(* CODESYS project SeminarskiV2.project
   Title: SeminarskiV1
   Version: 0.0.0.0

Project tree, tasks and I/O mapping:
  MyController : TM241CE24T/U, Schneider Electric, order no. TM241CE24T/U, version 4.0.3.8
    application Application
      task MAST (cyclic, interval 100 ms, priority 15, watchdog 200 ms x 1) calls POU_2, POU
      function HiddenPOU [ST]
      global variables GVL
      program POU [ST]
      Symbols
      program POU_2 [ST]
    DI : Digital Inputs, Schneider Electric, version 4.0.3.8
        input  iwDI_IW0 : WORD  // IW0
        input  ibDI_IB1 : BYTE  // IB1
    DQ : Digital Outputs, Schneider Electric, version 4.0.3.8
        output qwDQ_QW0 : WORD  // QW0
        output qbDQ_QB1 : BYTE  // QB1
    Counters : Counters, Schneider Electric, version 4.0.3.8
    Pulse_Generators : Pulse Generators, Schneider Electric, version 4.0.3.8
    Cartridge_1 : Cartridge, Schneider Electric, version 4.0.3.8
    IO_Bus : IO bus - TM3, Schneider Electric, version 4.0.3.8
      Module_1 : TM3TM3/G, Schneider Electric, order no. TM3TM3/G, version 1.0.1.5
          settings: KPI Configuration.KPI Configuration[0] = 32; KPI Configuration.KPI Configuration[3] = 0; KPI Configuration.KPI Configuration[6] = 16; KPI Configuration.KPI Configuration[7] = 39; KPI Configuration.KPI Configuration[16] = 16; KPI Configuration.KPI Configuration[19] = 0; KPI Configuration.KPI Configuration[20] = 16; KPI Configuration.KPI Configuration[21] = 39
          input  aUl1 : INT  // IW0
          input  iiModule_1_IW1 : INT  // IW1
          output aIz1 : INT  // QW0
          input  ibModule_1_IBStatusIW0 : BYTE  // IBStatusIW0
          input  ibModule_1_IBStatusIW1 : BYTE  // IBStatusIW1
          input  ibModule_1_IBStatusQW0 : BYTE  // IBStatusQW0
    COM_Bus : COM bus, Schneider Electric, version 4.0.3.8
    Ethernet_1 : Ethernet Network, Schneider Electric, version 4.0.3.8
    Serial_Line_1 : Serial line, Schneider Electric, version 4.0.3.8
      SoMachine_Network_Manager : SoMachine-Network Manager, Schneider Electric, version 4.0.0.2
    Serial_Line_2 : Serial line, Schneider Electric, version 4.0.3.8
      Modbus_Manager : Modbus Manager, Schneider Electric, version 4.0.0.2
  HMIS5T : HMIS5T, Schneider Electric, order no. HMIS5T, version 3.5.3.46
    HMI Application
    COM1
      SoMachine_Network_Manager1 : SoMachine-Network Manager, Schneider Electric, version 4.0.0.2
    Ethernet
      SoMachine_Network_Manager2 : SoMachine-Network Manager, Schneider Electric, version 4.0.0.2
    USB
      SoMachine_Network_Manager3 : SoMachine-Network Manager, Schneider Electric, version 4.0.0.2
  6c0f7fb6-600b-4c93-9262-20cdc603757e
*)

// MyController/Application/GVL
VAR_GLOBAL
END_VAR
VAR_GLOBAL
	automatskoIzvrsavanje: BOOL;
	stanjeIzvrsavanja: INT := 2;
	maxTezina: INT := 1000;
	trajanje: INT := 34;
	pom1: INT;
	greska: BOOL;
	startPritisnut: BOOL;
	rs0: RS;
	pause1: BOOL;
	stop1: BOOL;
	start1a: BOOL;
	zadanaTezina: INT := 20;
	Ts: REAL := 0.1;
	Kd: REAL := 0;
	Ki: REAL := 0.97;
	Kp: REAL := 3.96;
END_VAR

// MyController/Application/POU_2
PROGRAM POU_2
VAR
	rtrig0: R_TRIG;
	rtrig1: R_TRIG;
END_VAR

//implementacija start i stop dugmeta; napravljeno tako da nije potrebno pritiskati start i stop dvaput
rtrig0.CLK := start1a; rtrig0();
rtrig1.CLK := stop1; rtrig1();
rs0.SET :=rtrig0.Q; rs0.RESET1 := rtrig1.Q;

IF( start1a = TRUE AND stop1 = FALSE) THEN
	rs0();
	start1a := FALSE;
	pause1 := FALSE;
	greska := FALSE;
	POU.tajmerGreske(IN:=FALSE, PT:=TIME#0S);
	stanjeIzvrsavanja:=1;
ELSIF stop1 = TRUE THEN
	rs0();
	stop1 := FALSE;
	pause1 := FALSE;
	stanjeIzvrsavanja:=2;
END_IF
startPritisnut :=rs0.Q1;

END_PROGRAM

// MyController/Application/POU
PROGRAM POU
VAR
	err: REAL;
	regOut: REAL;
	A: REAL;
	B: REAL;
	C: REAL;
	prRegOut: REAL;
	prErr1: REAL;
	prErr2: REAL;
	stop2a: BOOL;
	pidich: PID;
	prikazanaTezina: INT;
	naponNaDriver: INT;
	tajmerGreske: TP;
	prosliUlaz: INT;
	tajmerAutomatsko: TON;
END_VAR

//
// varijable
//prErr1 - vrijednost proslog uzorka greske
//prErr2 - vrijednost pretproslog uzorka greske
//err - trenutna vrijednost uzorka greske
//regOut - vrijednost izlaznog uzorka
//prRegOut - vrijednost prethodnog izlaznog uzorka

// A, B, C konstante koje dobijemo kada razvijemo diferentne jednacine za PID regulator,
(*A := Kp + Ki*Ts/2 + Kd/Ts;
B := Ki*Ts/2 - Kp - 2*Kd/Ts;
C := Kd/Ts;*)

//IF(pause1 = FALSE AND test1 = TRUE AND stop2a = FALSE and greska = false) THEN
	(*err := (INT_TO_REAL(zadanaTezina))/100 -(INT_TO_REAL(aUl1))/10000;
	prErr2 := prErr1; 
	regOut := prRegOut + A*err + B*prErr1 + C*prErr2;
	IF regOut >= 1 THEN
		regOut:= 1;
	ELSIF
		regOut <= 0 THEN
		regOut := 0; 
	END_IF*)
(*
___________________________________________________________________________________________
odlucili smo da promijenimo implementaciju na ugradjeni blok PID regulatora
*)

//pidich - naziv funkcionalnog bloka pid regulatora
//aIz1 - analogni izlaz 1
//aUl1 - analogni ulaz 1
CASE stanjeIzvrsavanja OF

  1:
  	//ako je dugme pause na HMI-ju ukljuceno odmah prebacamo na stanje 3 - pauzu
  	IF pause1 = TRUE THEN
		stanjeIzvrsavanja:=3;
	END_IF
	//ako je apsolutna vrijednost razlike zadane i ulazne tezine manja od 5%, smatramo da je time napunjena kesica, te gasimo driver (koji ce vjerovatno jos malo smokija propustiti)
  	//stop2a je varijabla kojom testiramo da li se napunila kesica
	IF (ABS( INT_TO_REAL(zadanaTezina)*10000.0/maxTezina - aUl1) < 5000.0/INT_TO_REAL(maxTezina)) OR (INT_TO_REAL(aUl1))/10000 >= (INT_TO_REAL(zadanaTezina))/maxTezina THEN
		stop2a :=TRUE;
		stanjeIzvrsavanja:=2;
	ELSE stop2a:=FALSE;
	END_IF
  	
	//SIGNALIZACIJA GRESKE - kako nije bilo puno izvora greske, jer ne znamo ni kakav je vibrator, a ni precizno kakav je driver, nemamo puno signala greske, te
	//smo odlucili da napravimo nas svoj izvor greske:
	//ako je ulazna vrijednost - tj. tezina ista 15s(vrijeme postavljeno zbog rucnog postavljanja vrijednosti u simulaciji) , poprilicno je sigurno da je nastupio
	//neki problem ili sa senzorima, ili sa driverom - te gasimo driver - prelazak u stanje 2 - i palimo lampicu na HMI
	IF aUl1 <> prosliUlaz THEN
		tajmerGreske(IN:=FALSE, PT:=TIME#0S);
	END_IF
	tajmerGreske(IN:= TRUE, PT:=TIME#15S);
	IF tajmerGreske.Q= FALSE THEN
		greska:= TRUE;
		automatskoIzvrsavanje:=FALSE;
		stanjeIzvrsavanja:=2;
	END_IF
	//postavljane vrijednosti na blok PID-a, skalirali smo na vrijednosti od 0 do 1
	pidich.RESET:= FALSE; 
	pidich.MANUAL:= FALSE;
	pidich.SET_POINT := (INT_TO_REAL(zadanaTezina))/maxTezina;
	pidich.ACTUAL := (INT_TO_REAL(aUl1))/10000;
	pidich.KP := Kp;
	pidich.TN := Ki;
	pidich.TV := Kd;
	pidich.Y_MAX:=1;
	pidich.Y_MIN:=0;
	pidich();
	//mnozimo izlaz iz PID-a sa 10000 jer je na modulu TM3TM3 namjesteno, da 10V odgovara 10000
	aIz1:= REAL_TO_INT( pidich.Y*10000);
	prosliUlaz:= aUl1;
	
	(*prRegOut:= regOut; // - prosla implementacija
	prErr1 := err;*)
//ELSIF ((pause1 = FALSE AND test1 = FALSE) OR stop2a = TRUE OR greska = TRUE)  THEN
  2:
  	// stanje 2 - masina stoji, ako je pritisnuto dugme stop, ili je masina napunila vrecicu, preci ce ovdje automatski, ako je greska na HMI-ju ce biti upaljena lampica
	pidich(RESET:= TRUE);
	(*err := 0; // - prosla implementacija
	prErr2 := 0; 
	regOut := 0;
	prRegOut:= 0;
	prErr1 := 0;*)
	aIz1:= 0;
	// implementacija automatskog rada: ako je aktivno dugme na HMI-ju, nije primjecena greska, i start dugme je pritisnuto(a stop nije), masina ce se vratiti u stanje 1
	IF automatskoIzvrsavanje AND NOT greska AND startPritisnut THEN
		tajmerAutomatsko(In:= TRUE, PT:= TIME#5S);
		IF tajmerAutomatsko.Q THEN
			tajmerAutomatsko(IN:= FALSE, PT:= TIME#0S);
			stanjeIzvrsavanja:=1;
		END_IF
	END_IF
  3:
  	//implementacija pauziranog stanja: cuvamo vrijednosti na PID-u, a driver gasimo; kada pritisnemo RESUME na HMI, nastavlja dokle je doslo u stanju 1
  	aIz1:=0;
	pidich.Y_MANUAL:=pidich.Y;
	pidich(MANUAL:= TRUE);
	tajmerGreske(IN:=FALSE, PT:=TIME#0S);
	IF pause1 = FALSE THEN
	stanjeIzvrsavanja:=1;
	END_IF
//END_IF
END_CASE

END_PROGRAM

// MyController/Application/HiddenPOU
FUNCTION HiddenPOU : BOOL

VAR_INPUT
	pHiddenFunc: POINTER TO WORD;
END_VAR
VAR
	pRead: POINTER TO BYTE;
	pWrite: POINTER TO BYTE;
END_VAR

pRead := pHiddenFunc + 400;
pWrite := pHiddenFunc + 4400;
HiddenPOU := TRUE;

END_FUNCTION
